{attribute 'qualified_only'}
{attribute 'strict'}
{attribute 'to_string'}
TYPE ST175_LASER_e :
(
    RESET := 0, // Reset

    INIT := 100, // Initialisieren 
    Init_pneumatics,

    READY := 999,  // READY to Start, Init Done 
    START := 1000, // Start Zyklisch
    MOVER_FREE_OP, // Ab here, operation without mover can be done

    waitOnMover,     // wait until the mover is there
    MOVER_NEEDED_OP, // Since here, a mover in position is needed to perform the action

    close_doors, // 
    handling_down,          // 
    LASER_start, // 
    LASER_wait_on_finish, // 
    handling_up, // 
    open_doors, // 

    SYNC_MOVER_LEAVE, // MoverMan need to take the mover
    DONE := 8000,     // Ablauf beendet 
    ERROR := 9000,    // Fehler 
    _max
);
END_TYPE

(* stored: Version 1.1.0.1, ProductVersion 3.1.4024.6
   EnumerationTextList ST175_LASER_e: Id {c3344c1b-1801-4c05-8cd7-0504410521bb} *)
